Fanuc KAREL source: kd00058.KL

-- PROVISIONAL review KL for V770-1; original PC SHA256 fcb444d6732eb9b80415ab31a26ace6bad88ea4c5eaf51abae2d5e1d8f9aaa50
-- Incomplete behavior may be omitted. Consult companion uncertainty JSON. Do not deploy.
PROGRAM KD00058
%NOLOCKGROUP
VAR
  I : INTEGER
  J : INTEGER
  B : BOOLEAN
  R : REAL
  S : STRING[80]
BEGIN
  -- UNRESOLVED_PC offsets 5-18; opcodes 9D,81,18,9D,1B,9D,12,9C,13,04
  -- UNRESOLVED_PC offsets 23-27; opcodes 7F
END KD00058
